{attribute 'GeneratedUsingTerminal: EL6201-0000-0017'}
{attribute addProperty BoxType "EL6201-0000-0017"}
{attribute addProperty Id "Slave_2A_DO0BOOL1Slave_2A_DO1BOOL1Slave_2A_DO2BOOL1Slave_2A_DO3BOOL1Slave_2B_DO0BOOL1Slave_2B_DO1BOOL1Slave_2B_DO2BOOL1Slave_2B_DO3BOOL1"}
{attribute addProperty CRC "4010093849"}
{attribute addProperty Size "8"}
TYPE Slave_2_Outputs_EF052D19 :
STRUCT
	{attribute addProperty Name "Slave_2A_DO0"}
	Slave_2A_DO0 : BOOL;
	{attribute addProperty Name "Slave_2A_DO1"}
	Slave_2A_DO1 : BOOL;
	{attribute addProperty Name "Slave_2A_DO2"}
	Slave_2A_DO2 : BOOL;
	{attribute addProperty Name "Slave_2A_DO3"}
	Slave_2A_DO3 : BOOL;
	{attribute addProperty Name "Slave_2B_DO0"}
	Slave_2B_DO0 : BOOL;
	{attribute addProperty Name "Slave_2B_DO1"}
	Slave_2B_DO1 : BOOL;
	{attribute addProperty Name "Slave_2B_DO2"}
	Slave_2B_DO2 : BOOL;
	{attribute addProperty Name "Slave_2B_DO3"}
	Slave_2B_DO3 : BOOL;
END_STRUCT
END_TYPE

(* stored: Version 1.2.0.0, ProductVersion 3.1.4024.9
   DUT Slave_2_Outputs_EF052D19: Id {212dd07b-c652-4ac7-bd88-aea3059e1226} *)
